PROGRAM PnID
VAR_INPUT
	CircularPumpFlow AT %I*: INT;
	bHI AT %I*: BOOL;
	bLO AT %I*: BOOL;
END_VAR
VAR_OUTPUT
	bMotor1 AT %Q*: BOOL;
	bMotor2 AT %Q*: BOOL;
END_VAR
VAR
	ForceFan1: aFb_Motor;
	ForceFan2: aFb_Motor;
	ForceFan3: aFb_Motor;
	CondensePump: aFb_Motor;
	SupplyPump: aFb_Motor;
	CircularPump: aFb_Motor;
	InterPump: aFb_Motor;
	LPHeaterValve: aFb_Valve;
	AirEjectorValve: aFb_Valve;
	HPHeaterValve: aFb_Valve;
	TurbineValve: aFb_Valve;
	
	CirPumpFlowT: INT;
	temp: REAL;
END_VAR

//Control all components in the P&ID 

//Resolve Flow Sensor
CirPumpFlowT:= CircularPumpFlow;
temp := (INT_TO_REAL(CirPumpFlowT) - 630)*0.0006;
IF temp < 0 THEN
	Streams.OutStream.CircularPump_OutFlow := 0;
ELSE
	Streams.OutStream.CircularPump_OutFlow := temp;
END_IF

//Pumps
{region "Condense Pump"}
CondensePump(RunCondition := AutoControl.CondensePump_Press.Start,
				StopCondition := AutoControl.CondensePump_Press.Stop,
				SpeedCondition := AutoControl.CondensePump_Press.ControlSignal,
				RunFeedback := CondensePump.Cmd,
				Maxspeed := Interfacex.Parameters.MaxSpeed_CondensePump,//.MaxSpeed_CondensePump,
				ActualSpeed := Streams.InStream.CondensePump_Speed ,
				Speed => Streams.OutStream.CondensePump_SetSpeed,
				DisplayName := 'Condense Pump');
{endregion}
{region "Supply Pump"}
SupplyPump(RunCondition := AutoControl.SupplyPump_Press.Start,
				StopCondition := AutoControl.SupplyPump_Press.Stop,
				SpeedCondition := AutoControl.SupplyPump_Press.ControlSignal,
				RunFeedback := SupplyPump.Cmd,
				Maxspeed := Interfacex.Parameters.MaxSpeed_SupplyPump,
				ActualSpeed := Streams.InStream.SupplyPump_Speed,
				Speed => Streams.OutStream.SupplyPump_SetSpeed,
				DisplayName := 'Supply Pump');
{endregion}
	 
{region "Circular Pump"}
CircularPump(RunCondition := AutoControl.Condenser_Temp.Start,
				StopCondition := AutoControl.Condenser_Temp.Stop,
				SpeedCondition := Interfacex.Parameters.MaxSpeed_CircularPump,
				RunFeedback := CircularPump.Cmd,
				Maxspeed := Interfacex.Parameters.MaxSpeed_CircularPump,
				ActualSpeed := CircularPump.Speed,
				Cmd => bMotor2,
				DisplayName := 'Circular Pump');
{endregion}
	 
{region 'Intermediate Pump'}
InterPump(RunCondition := AutoControl.InterTank_Level.Start,
				StopCondition := AutoControl.InterTank_Level.Stop,
				SpeedCondition := Interfacex.Parameters.MaxSpeed_InterPump,
				RunFeedback := InterPump.Cmd,
				Maxspeed := Interfacex.Parameters.MaxSpeed_InterPump,
				ActualSpeed := InterPump.Speed,
				Cmd => bMotor1,
				DisplayName := 'Intermediate Pump');
{endregion}


//Valves
{region "Low Pressure Heater Valve"}
LPHeaterValve(RunCondition := AutoControl.LPHeater_Temp.Start,
				StopCondition := AutoControl.LPHeater_Temp.Stop,
				PercentCondition := AutoControl.LPHeater_Temp.ControlSignal,
				RunFeedback := LPHeaterValve.Cmd,
				OpenPercent => Streams.OutStream.LPHeaterValve_SetPercent,
				DisplayName := 'Low Pressure Heater Valve');
{endregion}
	 
{region "Deaerator"}
AirEjectorValve(RunCondition := AutoControl.AirEjector_Temp.Start,
				StopCondition := AutoControl.AirEjector_Temp.Stop,
				PercentCondition := AutoControl.AirEjector_Temp.ControlSignal,
				RunFeedback := AirEjectorValve.Cmd,
				OpenPercent => Streams.OutStream.AirEjectorValve_SetPercent,
				DisplayName := 'Deaerator Valve');
{endregion}
{region "High Pressure Heater Valve"}
HPHeaterValve(RunCondition := AutoControl.HPHeater_Temp.Start,
				StopCondition := AutoControl.HPHeater_Temp.Stop,
				PercentCondition := AutoControl.HPHeater_Temp.ControlSignal,
				RunFeedback := HPHeaterValve.Cmd,
				OpenPercent => Streams.OutStream.HPHeaterValve_SetPercent,
				DisplayName := 'High Pressure Heater Valve');
{endregion}
{region "Turbine Valve"}
TurbineValve(RunCondition := AutoControl.Turbine_Speed.Start,
				StopCondition := AutoControl.Turbine_Speed.Stop,
				PercentCondition := AutoControl.Turbine_Speed.ControlSignal,
				RunFeedback := TurbineValve.Cmd,
				OpenPercent => Streams.OutStream.TurbineValve_SetPercent,
				DisplayName := 'Turbine Valve');
{endregion}


//Fans
{region "ForceFan1"}
ForceFan1(RunCondition := AutoControl.Boiler_Temp.Start,
				StopCondition := AutoControl.Boiler_Temp.Stop,
				SpeedCondition := AutoControl.Boiler_Temp.ControlSignal,
				RunFeedback := ForceFan1.Cmd,
				Maxspeed := Interfacex.Parameters.MaxSpeed_ForceFan1,
				ActualSpeed := Streams.InStream.ForceFan1_Speed,
				Speed => Streams.OutStream.ForceFan1_SetSpeed,
				DisplayName := 'Force Fan 1');
{endregion}
	 
{region "ForceFan2"}
ForceFan2(RunCondition := AutoControl.Boiler_Temp.Start,
				StopCondition := AutoControl.Boiler_Temp.Stop,
				SpeedCondition := AutoControl.Boiler_Temp.ControlSignal,
				RunFeedback := ForceFan2.Cmd,
				Maxspeed := Interfacex.Parameters.MaxSpeed_ForceFan2,
				ActualSpeed := Streams.InStream.ForceFan2_Speed,
				Speed => Streams.OutStream.ForceFan2_SetSpeed,
				DisplayName := 'Force Fan 2');
{endregion}
{region "ForceFan3"}
ForceFan3(RunCondition := AutoControl.Boiler_Temp.Start,
				StopCondition := AutoControl.Boiler_Temp.Stop,
				SpeedCondition := AutoControl.Boiler_Temp.ControlSignal,
				RunFeedback := ForceFan3.Cmd,
				Maxspeed := Interfacex.Parameters.MaxSpeed_ForceFan3,
				ActualSpeed := Streams.InStream.ForceFan3_Speed,
				Speed => Streams.OutStream.ForceFan3_SetSpeed,
				DisplayName := 'Force Fan 3');
{endregion}

END_PROGRAM

(* stored: Version 1.1.0.1, ProductVersion 3.1.4024.4
   POU PnID: Id {10f77e3b-7018-4648-a34b-0c0909467aaf}, SpecialFunc None *)
